    30: (* Get reply *)
        fbReceiveData(
            pPrefix:=ADR(bDelimiter),
            LenPrefix:=1,
            pSuffix:=ADR(bDelimiter),
            LenSuffix:=1,
            pReceiveData:=ADR(baRxData),
            SizeReceiveData:=SIZEOF(baRxData),
            Timeout:= i_tTimeOut,
            Reset:= FALSE,
            RXbuffer:= iq_stSerialRXBuffer );
        tonTimeout(IN:= TRUE, PT:= i_tTimeOut);
        IF fbReceiveData.Error <> 0 THEN
            q_sResult := CONCAT('In step 30 fbReceiveData resulted in error: ', INT_TO_STRING(fbReceiveData.Error));
            iStep := 9000;
        ELSIF fbReceiveData.RxTimeout OR tonTimeout.Q THEN
            q_sResult := 'Serial device failed to reply within timeout period';
            q_xTimeout := TRUE;
            iStep := 9000;
        ELSIF fbReceiveData.DataReceived THEN
            udiRxLen := fbReceiveData.LenReceiveData;
            // For troubleshooting, use this to capture a specific command message reply


            IF udiRxLen > 0 THEN
                //Remove the stuffing
                FOR iSeek:=1 TO UDINT_TO_INT(udiRxLen) DO
                    IF baRxData[iSeek]=16#7D THEN
                        fbShiftByteArray(ptArray:=ADR(baRxData), iSize:=256, iCurrIndex:=iSeek, iMessageLen:=UDINT_TO_INT(udiRxLen), iShift:=-1);
                        IF fbShiftByteArray.q_xError THEN
                            q_sResult:='Transaction failed in step 30, while removing the stuffing Hans dropped some on the floor, oh Hans!';
                            iStep:=9000;
                            RETURN; // this way we catch the problem
                            ELSE
                                //iSeek now points to the escaped byte, once again invert the fifth bit to recover
                                baRxData[iSeek]:=baRxData[iSeek] XOR 16#10;
                                //Reduce the message length by one byte
                                udiRxLen := udiRxLen - 1;
                        END_IF
                    END_IF
                END_FOR
                //Byte stuffing removed and cleared at this point
                //Could check the checksum here...
                //naaa
                //Determine the Rx data length
                bRxLen := baRxData[5];
                IF i_bCmd = bCatch and bRxLen > 0 THEN
                MEMCPY(destAddr:=ADR(q_baRxUnit), srcAddr:=ADR(baRxData), n:=udiRxLen);
                END_IF
                //Snag the state byte while we're here
                q_bState := baRxData[4];
                q_iRxLen := BYTE_TO_INT(bRxLen);
                //Memcpy ze' data, check if memcpy is successful (returns other than zero) or bRxLen is zero (which causes memcpy to return zero)
                IF UDINT_TO_BOOL(MEMCPY(srcAddr:=(ADR(baRxData)+5), destAddr:=ADR(q_baRxData), n:=BYTE_TO_UINT(bRxLen))) OR (bRxLen=0) THEN
                    q_sResult := 'Success';
                    iStep:=100;
                    //For debugging
                    //MEMCPY(destAddr:=ADR(q_abLastRxData[iDataRx,1]), srcAddr:=ADR(baRxData), n:=c_ArraySize);
                    //IF iDataRx = c_DebugArraySize THEN iDataRx := 1; ELSE iDataRx := iDataRx +1; END_IF
                ELSE
                    q_sResult := 'Memcpy step failed, expected some bytes but was NOT able to export them via memcpy, investigate transaction fb';
                    iStep := 9000;
                END_IF
            END_IF
        END_IF


    100: (* done *)
        q_xDone:=TRUE;
        IF  i_xExecute = FALSE THEN
            q_xDone:= FALSE;
            q_bState:=16#00;
            iStep := 0;
        END_IF

    9000:
        q_xError := TRUE;
END_CASE

END_FUNCTION_BLOCK

// POUs/Sensirion/fSHDLCChecksum
FUNCTION fSHDLCChecksum : BYTE
VAR_INPUT
    i_bAdr	:	BYTE;
    i_bCmd	:	BYTE;
    i_bLen	:	BYTE;
    i_pbaTxData	:	POINTER TO BYTE;
END_VAR
VAR
    iIndex	:	INT;
END_VAR

(* Checksum is calc like so
Sum all the bytes within the frame
Take the LSN ie. nibble of the result and invert it
*)

fSHDLCChecksum := i_bAdr + i_bCmd + i_bLen;

IF i_bLen > 0 THEN
FOR iIndex:=0 TO BYTE_TO_INT(i_bLen)DO
    fSHDLCChecksum := fSHDLCChecksum + i_pbaTxData^;
    i_pbaTxData := i_pbaTxData + 1;
END_FOR
END_IF

// Inverting LSN
fSHDLCChecksum := fSHDLCChecksum XOR 16#FF;

END_FUNCTION

// POUs/TEC/FB_TECDriver
FUNCTION_BLOCK FB_TECDriver

VAR_INPUT
    i_xExecute				: BOOL;					(* rising edge execute *)
    i_tTimeOut				: TIME := t#10s;  		(* Maximum wait time for reply *)
    i_stControl				: ST_TECControl;
END_VAR
VAR_OUTPUT
    q_xDone					: BOOL;
    q_xError				: BOOL;
    q_xWarning				: BOOL;					(* set in the event of an unexpected reply *)
    q_xTimeout				: BOOL;
    q_sResult				: STRING(255);
    q_sLastSentString		: ARRAY[1..40] OF STRING;				(* Last String Sent to Serial Device - for debugging *)
    q_sLastReceivedString	: ARRAY[1..40] OF STRING;				(* Last String Received from Serial Device - for debugging *)
    q_stStatus				: ST_TECStatus;
END_VAR
VAR_IN_OUT
    iq_stSerialRXBuffer 	: ComBuffer;
    iq_stSerialTXBuffer 	: ComBuffer;
END_VAR
VAR
    rtExecute				: R_TRIG;
    iStep					: INT;
    sSendData				: STRING;
    fbTECTransaction		: FB_TECTransaction;
    (*fbFormatString			: FB_FormatString;*)
    (*fbSplit					: FB_Split255;*)
    asReplyFields			: ARRAY[1..20] OF T_MaxString;
    wChecksum: WORD;
    rtStartIntegration: R_TRIG;
    rtEndReset: R_TRIG;

    sWorking: STRING;
    strResponseExpected: STRING;
    diWorking	:	DINT;
END_VAR

(* This function block performs serial communication with a TC-36-25 TEC Driver *)

(* rising edge trigger *)
rtExecute(CLK:= i_xExecute);
IF rtExecute.Q  THEN
    q_xDone	:= FALSE;
    q_xError := FALSE;
    q_xWarning := FALSE;
    q_xTimeout := FALSE;
    q_sResult:= '';
    fbTECTransaction( i_xExecute:= FALSE, iq_stSerialRXBuffer:= iq_stSerialRXBuffer, iq_stSerialTXBuffer:= iq_stSerialTXBuffer );  (* reset *)

    iStep := 10;
END_IF

CASE iStep OF
    0: (* idle *)
        ;

    10: (* Get Current Temperature *)
        fbTECTransaction(
            i_xExecute:= TRUE,
            i_sAddress:=i_stControl.sAddress,
            i_sCmd:= '01',
            i_diParameter := 0,
            i_tTimeOut:= i_tTimeOut,
            iq_stSerialRXBuffer:= iq_stSerialRXBuffer,
            iq_stSerialTXBuffer:= iq_stSerialTXBuffer,
            i_CmdFlag :=FALSE);

        IF fbTECTransaction.q_xError THEN
            q_sResult := CONCAT('in Step 10 serial transaction failed with message: ', fbTECTransaction.q_sResult);
            iStep := 9000;
        ELSIF fbTECTransaction.q_xDone THEN
            q_stStatus.sReply := fbTECTransaction.q_sResponseData;
            sWorking :=LEFT(q_stStatus.sReply, 8);
            sWorking := CONCAT('16#', sWorking);
            q_stStatus.diTemp1 := STRING_TO_DINT(sWorking);
            fbTECTransaction( i_xExecute:= FALSE, iq_stSerialRXBuffer:= iq_stSerialRXBuffer, iq_stSerialTXBuffer:= iq_stSerialTXBuffer, i_CmdFlag :=FALSE);  (* reset *)
            iStep := 20;

        END_IF
    20: (* Read setpoint *)
        fbTECTransaction(
            i_xExecute:= TRUE,
            i_sAddress:=i_stControl.sAddress,
            i_sCmd:= '03', // command
            i_diParameter := 0, // always zero for query
            i_tTimeOut:= i_tTimeOut,
            iq_stSerialRXBuffer:= iq_stSerialRXBuffer,
            iq_stSerialTXBuffer:= iq_stSerialTXBuffer,
            i_CmdFlag :=FALSE);

        IF fbTECTransaction.q_xError THEN
            q_sResult := CONCAT('in Step 20 serial transaction failed with message: ', fbTECTransaction.q_sResult);
            iStep := 9000;
        ELSIF fbTECTransaction.q_xDone THEN
            q_stStatus.sReply := fbTECTransaction.q_sResponseData;
            sWorking :=LEFT(q_stStatus.sReply, 8);
            sWorking := CONCAT('16#', sWorking);
            q_stStatus.diSetPoint := STRING_TO_DINT(sWorking);
            fbTECTransaction( i_xExecute:= FALSE, iq_stSerialRXBuffer:= iq_stSerialRXBuffer, iq_stSerialTXBuffer:= iq_stSerialTXBuffer, i_CmdFlag :=FALSE);  (* reset *)
            iStep := 25;
        END_IF

    25: (* Read output ON/OFF *)
        fbTECTransaction(
            i_xExecute:= TRUE,
            i_sAddress:=i_stControl.sAddress,
            i_sCmd:= '46', // command
            i_diParameter := 0, // always zero for query
            i_tTimeOut:= i_tTimeOut,
            iq_stSerialRXBuffer:= iq_stSerialRXBuffer,
            iq_stSerialTXBuffer:= iq_stSerialTXBuffer,
            i_CmdFlag :=FALSE);

        IF fbTECTransaction.q_xError THEN
            q_sResult := CONCAT('in Step 25 serial transaction failed with message: ', fbTECTransaction.q_sResult);
            iStep := 9000;
        ELSIF fbTECTransaction.q_xDone THEN
            q_stStatus.sReply := fbTECTransaction.q_sResponseData;
            sWorking :=LEFT(q_stStatus.sReply, 8);
            sWorking := CONCAT('16#', sWorking);
            diWorking := STRING_TO_DINT(sWorking);
            q_stStatus.xOutputOn := DINT_TO_BOOL(diWorking);
            A_ResetTransaction();
            iStep := 30;
        END_IF

    30: (* Read the alarm status *)
        fbTECTransaction(
            i_xExecute:= TRUE,
            i_sAddress:=i_stControl.sAddress,
            i_sCmd:= '05', // command
            i_diParameter := 0, // always zero for query
            i_tTimeOut:= i_tTimeOut,
            iq_stSerialRXBuffer:= iq_stSerialRXBuffer,
            iq_stSerialTXBuffer:= iq_stSerialTXBuffer,
            i_CmdFlag :=FALSE);

        IF fbTECTransaction.q_xError THEN
            q_sResult := CONCAT('in Step 10 serial transaction failed with message: ', fbTECTransaction.q_sResult);
            iStep := 9000;
        ELSIF fbTECTransaction.q_xDone THEN
            q_stStatus.sReply := fbTECTransaction.q_sResponseData;
            sWorking :=LEFT(q_stStatus.sReply, 8);
            sWorking := CONCAT('16#', sWorking);
            diWorking := STRING_TO_DINT(sWorking);

            //Alarm assignment
            q_stStatus.xHiTemp	:=	diWorking.0;
            q_stStatus.xLoTemp	:=	diWorking.1;
            q_stStatus.xLoTemp	:=	diWorking.2;
            q_stStatus.xOverCurrent	:=	diWorking.3;
            q_stStatus.xOpenInput1	:=	diWorking.4;
            q_stStatus.xOpenInput2	:=	diWorking.5;
            q_stStatus.xDriverLowVoltage	:=	diWorking.6;

            fbTECTransaction( i_xExecute:= FALSE, iq_stSerialRXBuffer:= iq_stSerialRXBuffer, iq_stSerialTXBuffer:= iq_stSerialTXBuffer, i_CmdFlag :=FALSE);  (* reset *)
            iStep := 40;
        END_IF

    40: (* Output Power *)
        fbTECTransaction(
            i_xExecute:= TRUE,
            i_sAddress:=i_stControl.sAddress,
            i_sCmd:= '02', // command
            i_diParameter := 0, // always zero for query
            i_tTimeOut:= i_tTimeOut,
            iq_stSerialRXBuffer:= iq_stSerialRXBuffer,
            iq_stSerialTXBuffer:= iq_stSerialTXBuffer,
            i_CmdFlag :=FALSE);

        IF fbTECTransaction.q_xError THEN
            q_sResult := CONCAT('in Step 10 serial transaction failed with message: ', fbTECTransaction.q_sResult);
            iStep := 9000;
        ELSIF fbTECTransaction.q_xDone THEN
            q_stStatus.sReply := fbTECTransaction.q_sResponseData;
            sWorking :=LEFT(q_stStatus.sReply, 8);
            sWorking := CONCAT('16#', sWorking);
            diWorking := STRING_TO_DINT(sWorking);

            q_stStatus.diPercentOut := (diWorking/511)*100; //in percentage

            fbTECTransaction( i_xExecute:= FALSE, iq_stSerialRXBuffer:= iq_stSerialRXBuffer, iq_stSerialTXBuffer:= iq_stSerialTXBuffer, i_CmdFlag :=FALSE);  (* reset *)
            iStep := 5000;
        END_IF

    5000: (* Change Setpoint *)
        IF q_stStatus.diSetpoint <> i_stControl.diTempSetpoint THEN

            fbTECTransaction(
                i_xExecute:= TRUE,
                i_sAddress:=i_stControl.sAddress,
                i_sCmd:= '1c', // command
                i_diParameter := i_stControl.diTempSetpoint,
                i_tTimeOut:= i_tTimeOut,
                iq_stSerialRXBuffer:= iq_stSerialRXBuffer,
                iq_stSerialTXBuffer:= iq_stSerialTXBuffer,
                i_CmdFlag :=TRUE);
            IF fbTECTransaction.q_xError THEN
                q_sResult := CONCAT('in Step 5000 serial transaction failed with message: ', fbTECTransaction.q_sResult);
                iStep := 9000;
            ELSIF fbTECTransaction.q_xDone THEN
                fbTECTransaction(
                     i_xExecute:= FALSE,
                    iq_stSerialRXBuffer:= iq_stSerialRXBuffer,
                    iq_stSerialTXBuffer:= iq_stSerialTXBuffer,
                    i_CmdFlag:=FALSE );  (* reset *)
                iStep := 5010;
            END_IF
        ELSE
            iStep := 5010;
        END_IF

    5010: (* Output ON/OFF *)
        IF q_stStatus.xOutputOn <> i_stControl.xOutputOn THEN

            fbTECTransaction(
                i_xExecute:= TRUE,
                i_sAddress:=i_stControl.sAddress,
                i_sCmd:= '2d', // command
                i_diParameter := BOOL_TO_DINT(i_stControl.xOutputOn),
                i_tTimeOut:= i_tTimeOut,
                iq_stSerialRXBuffer:= iq_stSerialRXBuffer,
                iq_stSerialTXBuffer:= iq_stSerialTXBuffer,
                i_CmdFlag :=TRUE);
            IF fbTECTransaction.q_xError THEN
                q_sResult := CONCAT('in Step 5010 serial transaction failed with message: ', fbTECTransaction.q_sResult);
                iStep := 9000;
            ELSIF fbTECTransaction.q_xDone THEN
                fbTECTransaction(
                     i_xExecute:= FALSE,
                    iq_stSerialRXBuffer:= iq_stSerialRXBuffer,
                    iq_stSerialTXBuffer:= iq_stSerialTXBuffer,
                    i_CmdFlag:=FALSE );  (* reset *)
                iStep := 8000;
            END_IF
        ELSE
            iStep := 8000;
        END_IF


    8000: (* done *)
        q_xDone := TRUE;
        IF q_sResult = '' THEN
            q_sResult := 'Success';
            q_stStatus.xStatusValid := TRUE;
        END_IF
        IF  i_xExecute = FALSE THEN
            q_xDone:= FALSE;
            iStep := 0;
        END_IF

    9000:
        _A_ClearStatus();
        q_xTimeout := fbTECTransaction.q_xTimeout;
        q_xError := TRUE;
        q_stStatus.xStatusValid := FALSE;


END_CASE

q_sLastSentString := fbTECTransaction.q_sLastSentString;
q_sLastReceivedString := fbTECTransaction.q_sLastReceivedString;

ACTION _A_ClearStatus:
q_stStatus.sReply := '';
END_ACTION

ACTION A_ResetTransaction:
fbTECTransaction( i_xExecute:= FALSE, iq_stSerialRXBuffer:= iq_stSerialRXBuffer, iq_stSerialTXBuffer:= iq_stSerialTXBuffer, i_CmdFlag :=FALSE);  (* reset *)
END_ACTION

END_FUNCTION_BLOCK

// POUs/TEC/FB_TECTransaction
FUNCTION_BLOCK FB_TECTransaction
VAR_INPUT
    i_xExecute				: 	BOOL;				(* Rising edge execute *)
    i_sCmd					: 	STRING(2); 			(* Send Data *)
    i_sAddress				:	STRING(2);
    i_diParameter			:	DINT;
    i_tTimeOut				:	TIME := T#10S;  	(* Maximum wait time for reply *)
    i_CmdFlag: BOOL := FALSE;
END_VAR
VAR_OUTPUT
    q_xDone					: BOOL;
    q_sResponseData			: STRING;
    q_xError				: BOOL;
    q_xTimeout				: BOOL;
    q_sResult				: STRING;
    q_sLastSentString		: ARRAY[1..40] OF STRING;			(* Last String Sent to Serial Device - for debugging *)
    q_sLastReceivedString	: ARRAY[1..40] OF STRING;			(* Last String Received from Serial Device - for debugging *)
END_VAR
VAR_IN_OUT
    iq_stSerialRXBuffer 	: ComBuffer;
    iq_stSerialTXBuffer 	: ComBuffer;
END_VAR
VAR
    rtExecute				: R_TRIG;
    iStep					: INT;
    fbClearComBuffer		: ClearComBuffer;
    fbSendString			: SendString;
    fbReceiveString			: ReceiveString;
    sReceivedString			: STRING;
    tonTimeout				: TON;
    sSendString: STRING;
    iStringTx: INT := 1;
    iStringRx: INT := 1;

    iStringTxRx: INT := 1;
    sTxRxString: ARRAY[1..40] OF STRING;

    fbFormatParamString	:	FB_FormatString;
    fbFormatParamZPadString	:	FB_FormatString;
    fbFormatCSString	:	FB_FormatString;
    sParameter: STRING;
    iIndexChkSum: INT;
    wCsSum: WORD;
    udiParameter: UDINT;

END_VAR

(* This function block performs serial transactions with a TC-36-25 TEC Driver  *)

(* rising edge trigger *)
rtExecute(CLK:= i_xExecute);
IF rtExecute.Q THEN
    q_xDone	:= FALSE;
    q_sResponseData := '';
    q_xError := FALSE;
    q_xTimeout := FALSE;
    q_sResult:= '';
    q_sLastSentString[iStringTx] := '';
    q_sLastReceivedString[iStringRx]:= '';
    iStep := 10;
END_IF

CASE iStep OF
    0:
        ; (* idle *)

    10: (* clear com buffers *)
        fbClearComBuffer(Buffer:= iq_stSerialRXBuffer);
        fbClearComBuffer(Buffer:= iq_stSerialTXBuffer);
        (* Reset receive *)
        fbReceiveString(
            Reset:= TRUE,
            ReceivedString:= sReceivedString,
            RXbuffer:= iq_stSerialRXBuffer );
        (* build the string *)
        sSendString := CONCAT(i_sAddress, i_sCmd); (* adding the address and command/query *)
        IF i_CmdFlag THEN
            (* Convert the parameter into an 8-wide hex string twos complemented*)
            udiParameter := DINT_TO_UDINT(i_diParameter);
            fbFormatParamString(sFormat:= '%x', arg1:=F_UDINT(udiParameter)); // first convert to a string
            fbFormatParamZPadString(sFormat:='%08s', arg1:=F_STRING(fbFormatParamString.sOut));// then zero pad, because FB_Format string does not zero-pad hex strings naturally
            sParameter := fbFormatParamZPadString.sOut;
        ELSE
            sParameter := '00000000'; (* send zeros if we're querying *)
        END_IF
        (* Add parameter *)
        sSendString := CONCAT(sSendString, sParameter);

        (* Compute checksum *)
        A_Checksum();

        (* add stx at start *)
        sSendString := CONCAT('*', sSendString);
        (* append checksum *)
        fbFormatCSString(sFormat := '%02x', arg1:=F_WORD(wCsSum));
        sSendString	:= CONCAT(sSendString, fbFormatCSString.sOut);
         (*adding tail *)
        sSendString := CONCAT(sSendString,'$R'); (* add <cr> *)

        IF fbFormatParamString.bError OR fbFormatCSString.bError THEN
            q_sResult := CONCAT('In step 10 fbFormatString resulted in error: ', UDINT_TO_STRING(fbFormatParamString.nErrId));
            iStep := 9000;
        ELSE
            fbSendString( SendString:= sSendString, TXbuffer:= iq_stSerialTXBuffer );
        END_IF
        q_sLastSentString[iStringTx] := sSendString;
        IF iStringTx = 40 THEN iStringTx := 1; ELSE iStringTx := iStringTx +1; END_IF
        iStep := iStep + 10;

    20: (* Finish sending the String *)
        IF fbSendString.Busy THEN
            fbSendString( SendString:= sSendString, TXbuffer:= iq_stSerialTXBuffer );
        ELSIF fbSendString.Error <> 0 THEN
            q_sResult := CONCAT('In step 20 fbSendString resulted in error: ', INT_TO_STRING(fbSendString.Error));
            iStep := 9000;
        ELSIF NOT fbSendString.Busy THEN
            iStep:=iStep + 10;
        END_IF
        tonTimeout(IN:= FALSE);

    30: (* Get reply *)
        fbReceiveString(
            Prefix:= '*',
            Suffix:= '^',
            Timeout:= i_tTimeOut,
            Reset:= FALSE,
            ReceivedString:= sReceivedString,
            RXbuffer:= iq_stSerialRXBuffer );
        tonTimeout(IN:= TRUE, PT:= i_tTimeOut);
        IF fbReceiveString.Error <> 0 THEN
            q_sResult := CONCAT('In step 30 fbReceiveString resulted in error: ', INT_TO_STRING(fbReceiveString.Error));
            iStep := 9000;
        ELSIF fbReceiveString.RxTimeout OR tonTimeout.Q THEN
            q_sResult := 'Serial device failed to reply within timeout period';
            q_xTimeout := TRUE;
            iStep := 9000;
        ELSIF fbReceiveString.StringReceived THEN
            q_sLastReceivedString[iStringRx] := sReceivedString;
            IF iStringRx = 40 THEN iStringRx := 1; ELSE iStringRx := iStringRx +1; END_IF
            IF LEN(sReceivedString) < 2 THEN
                q_sResult := 'Reply too short.';
                iStep := 9000;
            ELSE
                (* Removing stx and ack *)
                q_sResponseData := LEFT(sReceivedString,LEN(sReceivedString)-1);
                q_sResponseData := RIGHT(q_sResponseData,LEN(q_sResponseData)-1);
                (* Checking for error messages *)
                IF q_sResponseData = 'XXXXXXXXc0' THEN
                        q_sResult := 'Checksum error reported by driver';
                        iStep := 9000;
                END_IF
                q_sResult := 'Success.';
                q_xDone:= TRUE;
                iStep := 100;
            END_IF
        END_IF




    100: (* done *)
        IF  i_xExecute = FALSE THEN
            q_xDone:= FALSE;
            iStep := 0;
        END_IF
        IF NOT i_CmdFlag THEN
            sTxRxString[iStringTxRx]:=CONCAT(CONCAT(q_sLastSentString[iStringTx], ' received '), q_sLastReceivedString[iStringRx]);
        END_IF
        IF iStringTxRx = 40 THEN iStringTxRx := 1; ELSE iStringTxRx := iStringTxRx +1; END_IF

    9000:
        q_xError := TRUE;;




END_CASE

ACTION A_Checksum:
wCsSum := 0;

FOR iIndexChkSum := 0 TO (LEN(sSendString) -1) DO
    wCsSum:= wCsSum + BYTE_TO_WORD(sSendString[iIndexChkSum]);
END_FOR
wCsSum	:= wCsSum MOD 256; (* modulo 256 *)
END_ACTION

END_FUNCTION_BLOCK

// POUs/TEST
PROGRAM TEST
VAR
{attribute 'pytmc' := 'pv: @(P):SEL:A'}
{attribute 'TcLinkTo' := '.stSensSerial.stComIn.Status := TIIB[M3 Selector A Serial IO (EP6002-0002)]^COM TxPDO-Map Inputs Channel 1^Status;
                          .stViciSerial.stComIn.Status := TIIB[M3 Selector A Serial IO (EP6002-0002)]^COM TxPDO-Map Inputs Channel 2^Status;
                          .stSensSerial.stComOut.Ctrl := TIID^MAIN (EtherCAT)^M3 Selector A Serial IO (EP6002-0002)^COM RxPDO-Map Outputs Channel 1^Ctrl;
                          .stViciSerial.stComOut.Ctrl := TIID^MAIN (EtherCAT)^M3 Selector A Serial IO (EP6002-0002)^COM RxPDO-Map Outputs Channel 2^Ctrl;
                          .stShaker01.q_xPwrDO := TIIB[M3 Selector A Digital IO (EP2338-1001)]^Channel 9^Output;
                          .stShaker02.q_xPwrDO := TIIB[M3 Selector A Digital IO (EP2338-1001)]^Channel 10^Output;
                          .stShaker03.q_xPwrDO := TIIB[M3 Selector A Digital IO (EP2338-1001)]^Channel 11^Output;
                          .stShaker04.q_xPwrDO := TIIB[M3 Selector A Digital IO (EP2338-1001)]^Channel 12^Output;
                          .stBaseIO.i_SyncUnitWC := TIID^MAIN (EtherCAT)^M3 Selector A (EP1111)^WcState^WcState;
'}
fbSelectorA : FB_SelectorM3;

{attribute 'pytmc' := 'pv: @(P):PCM:A'}
{attribute 'TcLinkTo' := '.stPropAir1.i_iPressRB := TIID^MAIN (EtherCAT)^PCM A (EP4374-0002)^AI Inputs Channel 1^Value;
                          .stPropAir2.i_iPressRB := TIID^MAIN (EtherCAT)^PCM A (EP4374-0002)^AI Inputs Channel 2^Value;
                          .stPropAir1.q_iPressCt := TIID^MAIN (EtherCAT)^PCM A (EP4374-0002)^AO Outputs Channel 3^Analog output;
                          .stPropAir2.q_iPressCt := TIID^MAIN (EtherCAT)^PCM A (EP4374-0002)^AO Outputs Channel 4^Analog output;
                          .stSerial1.stComIn.Status := TIID^MAIN (EtherCAT)^PCM A (EP6002-0002)^COM TxPDO-Map Inputs Channel 1^Status;
                          .stSerial2.stComIn.Status := TIID^MAIN (EtherCAT)^PCM A (EP6002-0002)^COM TxPDO-Map Inputs Channel 2^Status;
                          .stSerial1.stComOut.Ctrl := TIID^MAIN (EtherCAT)^PCM A (EP6002-0002)^COM RxPDO-Map Outputs Channel 1^Ctrl;
                          .stSerial2.stComOut.Ctrl := TIID^MAIN (EtherCAT)^PCM A (EP6002-0002)^COM RxPDO-Map Outputs Channel 2^Ctrl;
                          .stBaseIO.i_SyncUnitWC := TIID^MAIN (EtherCAT)^PCM A (EP1111)^WcState^WcState;
'}
fbPCMA		: FB_PressureControlModule;

{attribute 'pytmc' := 'pv: @(P):MAN'}
{attribute 'TcLinkTo' := '.stValve[1].qxDO := TIIB[Gas_Mani_ValveCtrl (EP2338-0001)]^Channel 9^Output;
                          .stValve[1].ixOPN := TIIB[Gas_Mani_ValveRbk (EP2338-0001)]^Channel 1^Input;
                          .stValve[2].qxDO := TIIB[Gas_Mani_ValveCtrl (EP2338-0001)]^Channel 10^Output;
                          .stValve[2].ixOPN := TIIB[Gas_Mani_ValveRbk (EP2338-0001)]^Channel 2^Input;
                          .stValve[3].qxDO := TIIB[Gas_Mani_ValveCtrl (EP2338-0001)]^Channel 11^Output;
                          .stValve[3].ixOPN := TIIB[Gas_Mani_ValveRbk (EP2338-0001)]^Channel 3^Input;
                          .stValve[4].qxDO := TIIB[Gas_Mani_ValveCtrl (EP2338-0001)]^Channel 12^Output;
                          .stValve[4].ixOPN := TIIB[Gas_Mani_ValveRbk (EP2338-0001)]^Channel 4^Input;
                          .stValve[5].qxDO := TIIB[Gas_Mani_ValveCtrl (EP2338-0001)]^Channel 13^Output;
                          .stValve[5].ixOPN := TIIB[Gas_Mani_ValveRbk (EP2338-0001)]^Channel 5^Input;
                          .stValve[6].qxDO := TIIB[Gas_Mani_ValveCtrl (EP2338-0001)]^Channel 14^Output;
                          .stValve[6].ixOPN := TIIB[Gas_Mani_ValveRbk (EP2338-0001)]^Channel 6^Input;
                          .stValve[7].qxDO := TIIB[Gas_Mani_ValveCtrl (EP2338-0001)]^Channel 15^Output;
                          .stValve[7].ixOPN := TIIB[Gas_Mani_ValveRbk (EP2338-0001)]^Channel 7^Input;
                          .stBaseIO.i_SyncUnitWC :=	TIID^MAIN (EtherCAT)^Gas_Mani (EP1111)^WcState^WcState;
'}
fbGasMan : FB_GasManifold;

{attribute 'pytmc' := 'pv: @(P):MFM:A'}
{attribute 'TcLinkTo' := '.stMFM.i_rFlow := TIID^MAIN (EtherCAT)^Bronkhorst MFM A^TxPDO Map^fMeasure;
                          .stMFM.q_rSetpoint := TIID^MAIN (EtherCAT)^Bronkhorst MFM A^RxPDO Map^fSetpoint;
'}
fbBronkhorstA : FB_BronkhorstMFM;

{attribute 'pytmc' := 'pv: @(P):SPR:A'}
{attribute 'TcLinkTo' := '.q_xDO1 := TIIB[Solenoid Pair A Digital IO (EP2338-0001)]^Channel 9^Output;
                          .q_xDO2 := TIIB[Solenoid Pair A Digital IO (EP2338-0001)]^Channel 10^Output;
'}
fbSolenoidPairA : FB_SolenoidPair;

END_VAR

fbSelectorA();
fbPCMA();
fbGasMan();
fbBronkhorstA();
fbSolenoidPairA();

(* Following execution of all the programs, set the first pass false *)
g_xFirstPass := FALSE;

END_PROGRAM
